Fanuc KAREL source: kd00033.KL

-- PROVISIONAL review KL for V1013-1; original PC SHA256 54eb17c3b3109aae097e503a30a56fa9dd0151581c237395e295d98c2b31bd16
-- Incomplete behavior may be omitted. Consult companion uncertainty JSON. Do not deploy.
PROGRAM KD00033
%NOLOCKGROUP
VAR
  I : INTEGER
  J : INTEGER
  B : BOOLEAN
  R : REAL
  S : STRING[80]
BEGIN
  -- UNRESOLVED_PC offsets 5-24; opcodes 9D,81,18,9D,1B,9D,12,22,9D,13,04
  -- UNRESOLVED_PC offsets 29-33; opcodes 7F
END KD00033
